(* PLC project Thermostat PID, Actility iec61131 1.0.28, author Laurent Nicq *)
(* stored: creationDateTime 2013-04-23T20:30:50, contentDescription Thermostat sample application using the PID defined in the IEC standard, version V1.0.0, modificationDateTime 2013-09-16T15:54:21 *)

FUNCTION_BLOCK PWM
  VAR_INPUT
    PWM2_Start : BOOL;
    PWM2_Period : TIME;
  END_VAR
  VAR
    PWM2_Running_ON_Time : TIME;
  END_VAR
  VAR_INPUT
    PWM2_Ratio : DINT;
  END_VAR
  VAR
    PWM2_Limit_Low : DINT := 0;
    PWM2_Limit_High : DINT := 100;  (* If not set as INPUT, put 100.0 as initial value *)
    PWM2_ResetMode : DINT := 0;  (* For simulation *)
  END_VAR
  VAR_OUTPUT
    PWM2_Out : BOOL;
  END_VAR
  VAR
    PWM_HEATING : PWM_GENERATOR;
  END_VAR

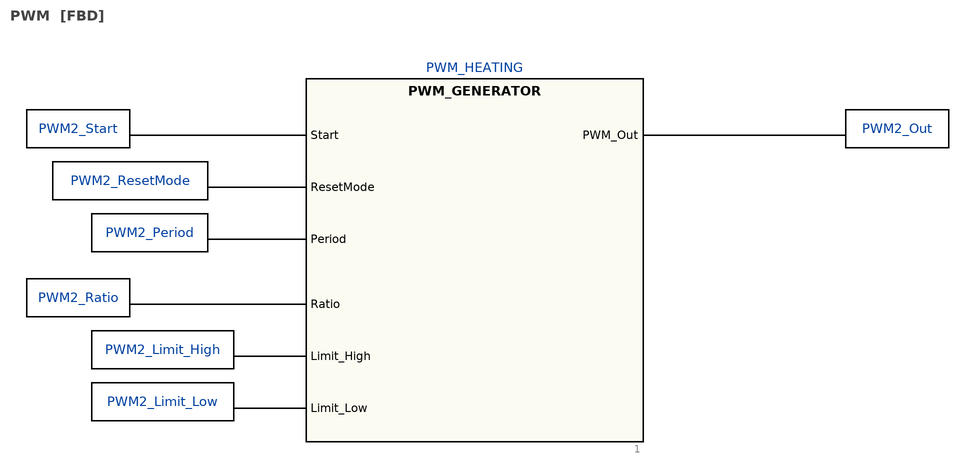
(* FBD diagram, written out as Structured Text *)
PWM_HEATING(Start := PWM2_Start, ResetMode := PWM2_ResetMode, Period := PWM2_Period, Ratio := PWM2_Ratio, Limit_High := PWM2_Limit_High, Limit_Low := PWM2_Limit_Low);
PWM2_Out := PWM_HEATING.PWM_Out;
END_FUNCTION_BLOCK

PROGRAM Thermostat_PID
  VAR
    TH_PWM_Period : TIME := T#20s;  (* Period in Second *)
    TH_PWM_Ratio : DINT;  (* from 0% to 100% *)
    TH_AUTO : BOOL := TRUE;  (* Thermostat mode *)
    TH_PWM_Start : BOOL := FALSE;  (* Needs RISING Edge to start *)
    TH_Setpoint : REAL := 28.0;
    TH_Room_Temperature : REAL := 25.0;
    TH_PROP : REAL := 0.5;
    TH_INTEGRAL : REAL := 0;
    TH_DERIVATE : REAL := 0;
    TH_Manual_Value : REAL := 0;  (* Value when AUTO is False *)
    TH_PID_Out : REAL := 0;  (* Value when AUTO is False *)
  END_VAR
  VAR_EXTERNAL
    TH_Relay_Output : BOOL;  (* PWM result *)
  END_VAR
  VAR
    TH_Cycle : TIME := T#1s;  (* Task Cycle *)
    PWM_For_Thermostat : PWM;
    PID_Test_Block : PID;
  END_VAR
  VAR  (* added by the conversion: wires and edge detectors of the diagram *)
    _MUL23_OUT : REAL;
    _REAL_TO_DINT26_OUT : DINT;
    _NOT13_OUT : BOOL;
  END_VAR

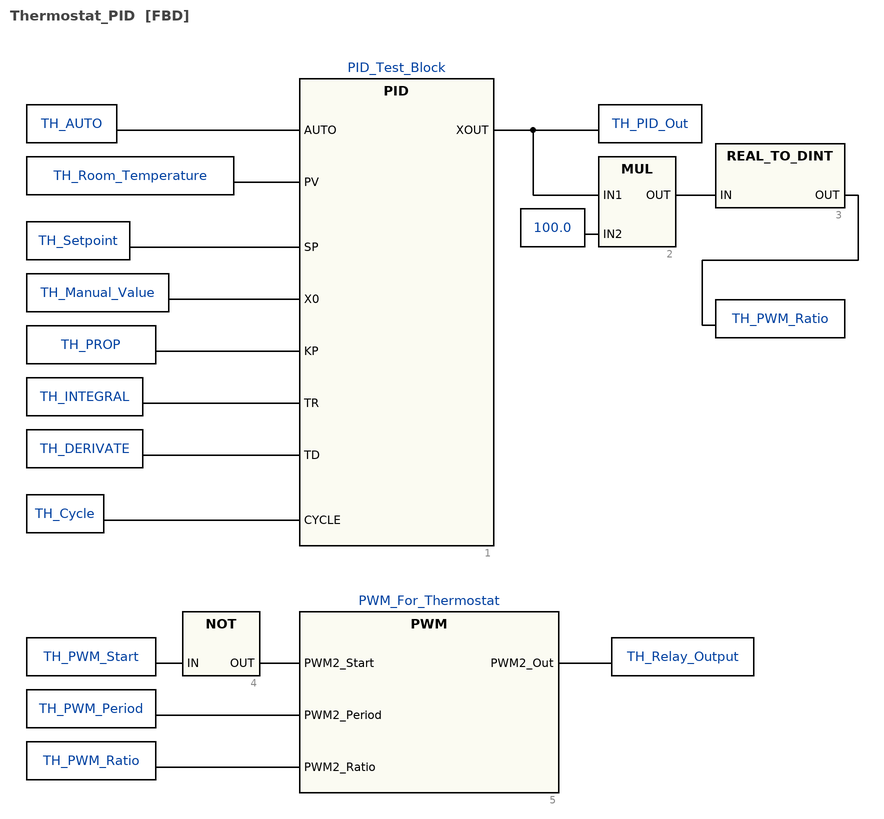
(* FBD diagram, written out as Structured Text *)
PID_Test_Block(AUTO := TH_AUTO, PV := TH_Room_Temperature, SP := TH_Setpoint, X0 := TH_Manual_Value, KP := TH_PROP, TR := TH_INTEGRAL, TD := TH_DERIVATE, CYCLE := TH_Cycle);
_MUL23_OUT := PID_Test_Block.XOUT * 100.0;
_REAL_TO_DINT26_OUT := REAL_TO_DINT(_MUL23_OUT);
_NOT13_OUT := NOT TH_PWM_Start;
PWM_For_Thermostat(PWM2_Start := _NOT13_OUT, PWM2_Period := TH_PWM_Period, PWM2_Ratio := TH_PWM_Ratio);
TH_PID_Out := PID_Test_Block.XOUT;
TH_PWM_Ratio := _REAL_TO_DINT26_OUT;
TH_Relay_Output := PWM_For_Thermostat.PWM2_Out;
END_PROGRAM

CONFIGURATION config
  RESOURCE Thermostat1 ON PLC
    VAR_GLOBAL
      TH_Room_Temperature_Sensor : REAL;
      TH_Relay_Output : BOOL;
    END_VAR
    TASK task1(INTERVAL := T#250ms, PRIORITY := 0);
    PROGRAM PID_Test WITH task1 : Thermostat_PID;
  END_RESOURCE
END_CONFIGURATION
